{attribute 'reflection'}
FUNCTION_BLOCK PUBLIC FB_DevAnalogInput EXTENDS FB_DevBase
VAR_INPUT
	bCmdSimulate	: BOOL 	:= FALSE ;// Simulate sensor Input 
	fSimValue		: INT	:= 0 ;// Simulated sensor state
END_VAR
VAR_OUTPUT
	fValue	: LREAL := 0 ; // Input value from hardware (converted to LREAL)
END_VAR
VAR
	inHwInput 	AT%I* : INT ; // Hardware connection
	inStatus	AT%I* : BYTE; // input card hardware status
END_VAR

// Set device type
eDevType := E_Devices.AnalogSensor ;

// Call base function
SUPER^();

// Check Hardware connection
CheckHardware();
// set feedback
ExecSetFeedback();

// Make sure compiler does not skip unused variables

METHOD CheckHardware : BOOL
VAR_INPUT
END_VAR
// Check for hardware faults
IF inStatus.0 THEN // signal under range
	stFault.Active			:= TRUE 							;
	stFault.Description		:= 'Signal under range';
	stFault.FaultType		:= E_FaultTypes.CF 					;
	bErrorActive			:= TRUE 							;
END_IF

IF inStatus.1 THEN // signal over range
	stFault.Active			:= TRUE 							;
	stFault.Description		:= 'Signal over range';
	stFault.FaultType		:= E_FaultTypes.CF 					;
	bErrorActive			:= TRUE 							;
END_IF

IF inStatus.6 THEN // general error bit
	stFault.Active			:= TRUE 							;
	stFault.Description		:= 'Hardware General Error';
	stFault.FaultType		:= E_FaultTypes.FF 					;
	bErrorActive			:= TRUE 							;
END_IF
END_METHOD

METHOD ExecSetFeedback : BOOL
VAR_INPUT
END_VAR
IF bCmdSimulate THEN 
	fValue := int_to_lreal(fSimValue) ;
ELSE
	fValue := INT_TO_LREAL(inHwInput);
END_IF

ExecSetFeedback := TRUE;
END_METHOD

METHOD PUBLIC Init : BOOL
VAR_INPUT
	// Location data for messages  
	nId			: UINT ; // Identification number of object
	nParentId	: UDINT ; // Id of higher level If aplicable (0 = no parent)
END_VAR
// ====== Set init to true =====
	bInitOk	:= TRUE ; 

// ====== Calculate device id =====
	bInitOk :=	ExecIdentifyDevice(nId,nParentId, E_ComponentTypes.AnInput) AND bInitOk;

// ====== Set feedback =====
	Init := bInitOk ;
END_METHOD

END_FUNCTION_BLOCK

(* stored: Version 1.1.0.1, ProductVersion 3.1.4024.11
   POU FB_DevAnalogInput: Id {438fca26-964b-0408-10a5-3e8ee84a0164}, SpecialFunc None
   Method CheckHardware: Id {a46229ba-2910-0c8c-007b-bec4165a24ff}
   Method ExecSetFeedback: Id {7a115a3e-3411-01c5-2bf8-56b6258af2f3}
   Method Init: Id {3357007e-f480-0c2c-080e-7ce021956725} *)
